Staubli VAL3: GetAxis7Pos.pgx

public program GetAxis7Pos(num& x_nPosition (dimensions=1), num x_nPrecent (dimensions=1))
begin

  dDio["O4_b7RecordPos"]=true
  delay(0.05)
  dDio["O4_b7RecordPos"]=false

  x_nPosition=aioGet(aAio["In4_a7CurPosH"])*power(2,16)+aioGet(aAio["In4_a7CurPosL"])
  x_nPosition=x_nPosition/max(x_nPrecent,0.001)

end
